FUNCTION_BLOCK MECH_HMIL (* HMI for testing MECH_VIEWL *)
  (* Standard: 61499-1; Classification: HMI; ApplicationDomain: SImulation *)
  (* Version 0.6, 2006-03-19, JHC, Holobloc Inc, Changed import to fb.rt.hmi *)
  (* Version 0.5, 2005-06-01, JHC, Holobloc Inc, Recompiled with new emitter. *)
  (* Version 0.4, 2005-06-01, JHC, Holobloc Inc, Recompiled with new emitter. *)
  (* Version 0.3, 2004-09-04, JHC, Rockwell Automation, Changed to optimized PUBL, standardized REND_ID. *)
  (* Version 0.2, 2002-05-02, JHC, Rockwell Automation, Changed to optimized PUBL, standardized REND_ID. *)
  (* Version 0.1, 2002-04-21, JHC, Rockwell Automation, Changed PUBL to PUBLISH *)
  (* Version 0.0, 2002-04-14, JHC, Rockwell Automation *)
  (* Compiler header: package fb.rt.mva; import fb.rt.hmi.*; import fb.rt.net.*; *)
  (* Compiler classdef: public class MECH_HMIL extends FBMVCD *)
  (* Compiler Java IBM VisualAge 3.0 *)
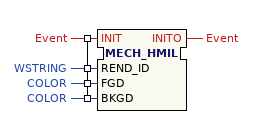
  EVENT_INPUT
    INIT WITH REND_ID, BKGD, FGD; (* Initialization Request *)
  END_EVENT
  EVENT_OUTPUT
    INITO; (* Initialization Confirm *)
  END_EVENT
  VAR_INPUT
    REND_ID : WSTRING; (* Data Channel ID - default is FB instaqnce name *)
    FGD : COLOR := red; (* Slider Foreground Color *)
    BKGD : COLOR := blue; (* Slider Background Color *)
  END_VAR
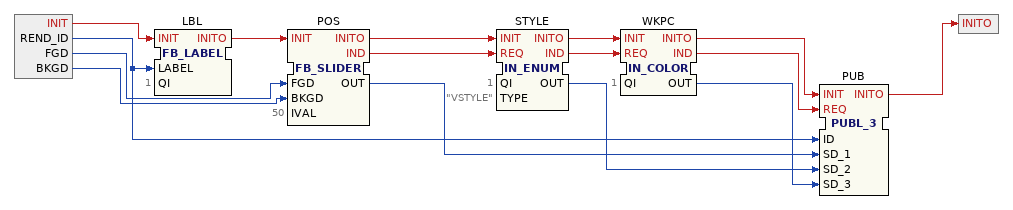
  FBS
    LBL : FB_LABEL(QI := 1);
    POS : FB_SLIDER(IVAL := 50);
    STYLE : IN_ENUM(QI := 1, TYPE := "VSTYLE");
    WKPC : IN_COLOR(QI := 1);
    PUB : PUBL_3;
  END_FBS
  EVENT_CONNECTIONS
    INIT TO LBL.INIT;
    LBL.INITO TO POS.INIT;
    POS.INITO TO STYLE.INIT;
    STYLE.INITO TO WKPC.INIT;
    WKPC.INITO TO PUB.INIT;
    PUB.INITO TO INITO;
    POS.IND TO STYLE.REQ;
    STYLE.IND TO WKPC.REQ;
    WKPC.IND TO PUB.REQ;
  END_CONNECTIONS
  DATA_CONNECTIONS
    REND_ID TO PUB.ID;
    REND_ID TO LBL.LABEL;
    POS.OUT TO PUB.SD_1;
    STYLE.OUT TO PUB.SD_2;
    WKPC.OUT TO PUB.SD_3;
    FGD TO POS.FGD;
    BKGD TO POS.BKGD;
  END_CONNECTIONS
END_FUNCTION_BLOCK
